FUNCTION_BLOCK SIMPLE_SLOT_ORIGIN_END_VECTORS_AND_CENTER (* Sets origin and end vectors for travel_path and also arc center for circular paths *)
  (* Standard: 61499-2 *)
  (* Version 1.0, 26-05-12, GASR, Universidade do Estado de Santa Catarina *)
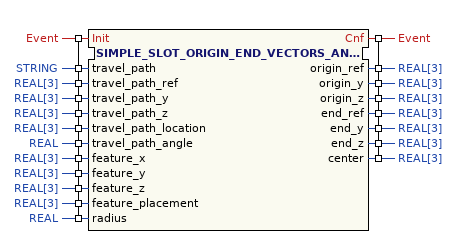
  EVENT_INPUT
    Init WITH travel_path, travel_path_ref, travel_path_y, travel_path_z, travel_path_location, travel_path_angle, feature_x, feature_y, feature_z, feature_placement, radius;
  END_EVENT
  EVENT_OUTPUT
    Cnf WITH origin_ref, origin_y, origin_z, end_ref, end_y, end_z, center;
  END_EVENT
  VAR_INPUT
    travel_path : STRING;
    travel_path_ref : ARRAY [0..2] OF REAL;
    travel_path_y : ARRAY [0..2] OF REAL;
    travel_path_z : ARRAY [0..2] OF REAL;
    travel_path_location : ARRAY [0..2] OF REAL;
    travel_path_angle : REAL;
    feature_x : ARRAY [0..2] OF REAL;
    feature_y : ARRAY [0..2] OF REAL;
    feature_z : ARRAY [0..2] OF REAL;
    feature_placement : ARRAY [0..2] OF REAL;
    radius : REAL;
  END_VAR
  VAR_OUTPUT
    origin_ref : ARRAY [0..2] OF REAL;
    origin_y : ARRAY [0..2] OF REAL;
    origin_z : ARRAY [0..2] OF REAL;
    end_ref : ARRAY [0..2] OF REAL;
    end_y : ARRAY [0..2] OF REAL;
    end_z : ARRAY [0..2] OF REAL;
    center : ARRAY [0..2] OF REAL;
  END_VAR
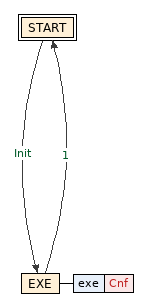
  EC_STATES
    START;
    EXE : exe -> Cnf;
  END_STATES
  EC_TRANSITIONS
    START TO EXE := Init;
    EXE TO START := 1;
  END_TRANSITIONS
  ALGORITHM exe IN Lua:
if( travel_path == 'LINEAR_PATH' ) then
	for i = 1, 3 do
		origin_ref[i] = travel_path_ref[i]
		origin_y[i] = travel_path_y[i]
		origin_z[i] = travel_path_z[i]
		end_ref[i] = travel_path_ref[i]
		end_y[i] = travel_path_y[i]
		end_z[i] = travel_path_z[i]
	end
    print( 'origin_ref before', origin_ref[1], origin_ref[2], origin_ref[3] )
    print( 'origin_y before', origin_y[1], origin_y[2], origin_y[3] )
    print( 'feature x', feature_x[1], feature_x[2], feature_x[3] )
    print( 'feature y', feature_y[1], feature_y[2], feature_y[3] )
    print( 'feature z', feature_z[1], feature_z[2], feature_z[3] )
	origin_ref = { origin_ref[1]*feature_x[1] + origin_ref[2]*feature_y[1] + origin_ref[3]*feature_z[1],
                   origin_ref[1]*feature_x[2] + origin_ref[2]*feature_y[2] + origin_ref[3]*feature_z[2],
                   origin_ref[1]*feature_x[3] + origin_ref[2]*feature_y[3] + origin_ref[3]*feature_z[3] }
	origin_y = { origin_y[1]*feature_x[1] + origin_y[2]*feature_y[1] + origin_y[3]*feature_z[1],
                 origin_y[1]*feature_x[2] + origin_y[2]*feature_y[2] + origin_y[3]*feature_z[2],
                 origin_y[1]*feature_x[3] + origin_y[2]*feature_y[3] + origin_y[3]*feature_z[3] }
    print( 'origin_ref', origin_ref[1], origin_ref[2], origin_ref[3] )
    print( 'origin_y', origin_y[1], origin_y[2], origin_y[3] )
elseif( travel_path == 'COMPLETE_CIRCULAR_PATH' ) then
	for i = 1, 3 do
		origin_ref[i] = travel_path_ref[i]
		origin_y[i] = travel_path_y[i]
		origin_z[i] = travel_path_z[i]
		end_ref[i] = travel_path_ref[i]
		end_y[i] = travel_path_y[i]
		end_z[i] = travel_path_z[i]
	end
	print( travel_path_z[1], travel_path_z[2], travel_path_z[3] )
	print( 'travel_path_location', travel_path_location[1] )
	center[1] = feature_placement[1] + ( travel_path_location[1]*feature_x[1] + travel_path_location[2]*feature_y[1] + travel_path_location[3]*feature_z[1] )
	center[2] = feature_placement[2] + ( travel_path_location[1]*feature_x[2] + travel_path_location[2]*feature_y[2] + travel_path_location[3]*feature_z[2] )
	center[3] = feature_placement[3] + ( travel_path_location[1]*feature_x[3] + travel_path_location[2]*feature_y[3] + travel_path_location[3]*feature_z[3] )
elseif( travel_path == 'PARTIAL_CIRCULAR_PATH' ) then
	for i = 1, 3 do
        origin_ref[i] = travel_path_ref[1]*feature_x[i] + travel_path_ref[2]*feature_y[i] + travel_path_ref[3]*feature_z[i]
        origin_y[i] = travel_path_y[1]*feature_x[i] + travel_path_y[2]*feature_y[i] + travel_path_y[3]*feature_z[i]
        origin_z[i] = travel_path_z[1]*feature_x[i] + travel_path_z[2]*feature_y[i] + travel_path_z[3]*feature_z[i]
    end
    print( 'vectors_start', origin_ref[1], origin_ref[2], origin_ref[3], origin_y[1], origin_y[2], origin_y[3], origin_z[1], origin_z[2], origin_z[3] )
	end_ref[1] = origin_ref[1]+math.cos( travel_path_angle*180/math.pi )
	end_ref[2] = origin_ref[2]+math.sin( travel_path_angle*180/math.pi )
	end_ref[3] = origin_ref[3]
	end_y[1] = -origin_y[1]+math.sin( travel_path_angle*180/math.pi )
	end_y[2] = origin_y[2]+math.cos( travel_path_angle*180/math.pi )
	end_y[3] = origin_y[3]
	print( 'vectors_end', end_ref[1], end_ref[2], end_ref[3], end_y[1], end_y[2], end_y[3], end_z[1], end_z[2], end_z[3] )
	center[1] = feature_placement[1] + ( travel_path_location[1]*feature_x[1] + travel_path_location[2]*feature_y[1] + travel_path_location[3]*feature_z[1] )
	center[2] = feature_placement[2] + ( travel_path_location[1]*feature_x[2] + travel_path_location[2]*feature_y[2] + travel_path_location[3]*feature_z[2] )
	center[3] = feature_placement[3] + ( travel_path_location[1]*feature_x[3] + travel_path_location[2]*feature_y[3] + travel_path_location[3]*feature_z[3] )
end
  END_ALGORITHM
END_FUNCTION_BLOCK
